PROGRAM FermentationProcess
VAR
	
(************** NAPĘDY **************************************************)
	fbDrv_MX01 		 : FB_Drive_1C();		//Napedy U11 mieszadła MX01	
	fbDrvContr_MX01  : FB_DriveControl(fbDrv_MX01);

	fbDrv_MX02 		 : FB_Drive_1C(); 		//Napedy U11 mieszadła MX01	
	fbDrvContr_MX02  : FB_DriveControl(fbDrv_MX02);

(************** Temp Sensor **************************************************)
	fbTempSens_T01	 : FB_Scaling; //Czujnik temperatury w reaktorze R01
	
(************** Ph Sensor **************************************************)
	fbPhSens_Ph01	 : FB_Scaling; //Czujnik ph w reaktorze R01

(************** Pressure Sensor **************************************************)
	fbPressureSens_P01	 : FB_Scaling; //Czujnik ciśnienia w reaktorze R01

(************** Hydrostatic pressure Sensor ************************************)
	fbHydrosPressureSens_HP01	  : FB_Scaling;
	
(************** Level Sensor **************************************************)
	fbLevelSens_L01	 : FB_Scaling; //Czujnik poziomu cieczy w reaktorze R01

(************** Reactor Mixers ***********************************************)
	fbReactorMixers	 : FB_ReactorMixer;	
	

END_VAR
VAR // added by the converter: edge detectors and wires of the graphical bodies
    _w1 : TIME;
    _w2 : ANY;
END_VAR

//Action
ACT_PhSens();       //skalowanie ph
ACT_PressureSens(); //skalowanie ciśnienie
ACT_TempSens();     //skalowanie temperatura
ACT_LevelSens();    //skalowanie poziom
ACT_Motor();    	//nastawy z SCADA
ACT_ReactorMixers();//Mieszanie w R01



//MX01
fbDrvContr_MX01();
GVL_Fermentation.stDriveStatus_MX01 := fbDrvContr_MX01.StatusStruct(); //zwróc strukturę

//MX02
fbDrvContr_MX02();
GVL_Fermentation.stDriveStatus_MX02 := fbDrvContr_MX02.StatusStruct(); //zwróc strukturę

ACTION ACT_LevelSens:
//Wyznacz poziom płynu w komorze fermentora zgodnie z wzorem (mH2O-P[kPa]*0.1)+poziom na ktorym wisi sonda hydrostatyczna
//przyjeto Ro =1kg/m3 g=9.81m2/s
GVL_Fermentation.LevelSens_R01.rValue := GVL_Fermentation.HydroPressSens_R01.rValue - GVL_Fermentation.PressureSens_R01.rValue * 0.1 + 0.12;
END_ACTION

ACTION ACT_Motor:
//Naped ustawienia MX01 i MX02
//nastawy z SCADA MX01
fbDrvContr_MX01.SetForward:=GVL_Fermentation.stDriveStatus_MX01.bForward;
//nastawy z SCADA MX02
fbDrvContr_MX02.SetForward:=GVL_Fermentation.stDriveStatus_MX02.bForward;
END_ACTION

ACTION ACT_PhSens:
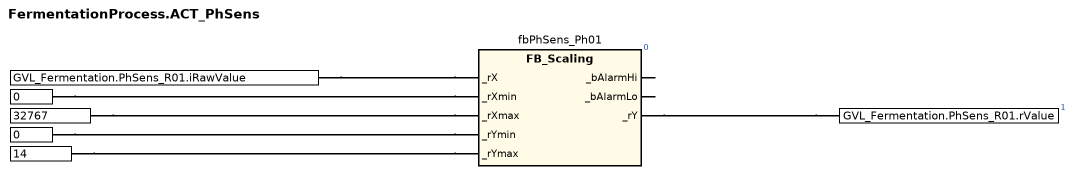
fbPhSens_Ph01(
    _rX := GVL_Fermentation.PhSens_R01.iRawValue,
    _rXmin := 0,
    _rXmax := 32767,
    _rYmin := 0,
    _rYmax := 14); // FB_Scaling
GVL_Fermentation.PhSens_R01.rValue := fbPhSens_Ph01._rY;
END_ACTION

ACTION ACT_PressureSens:
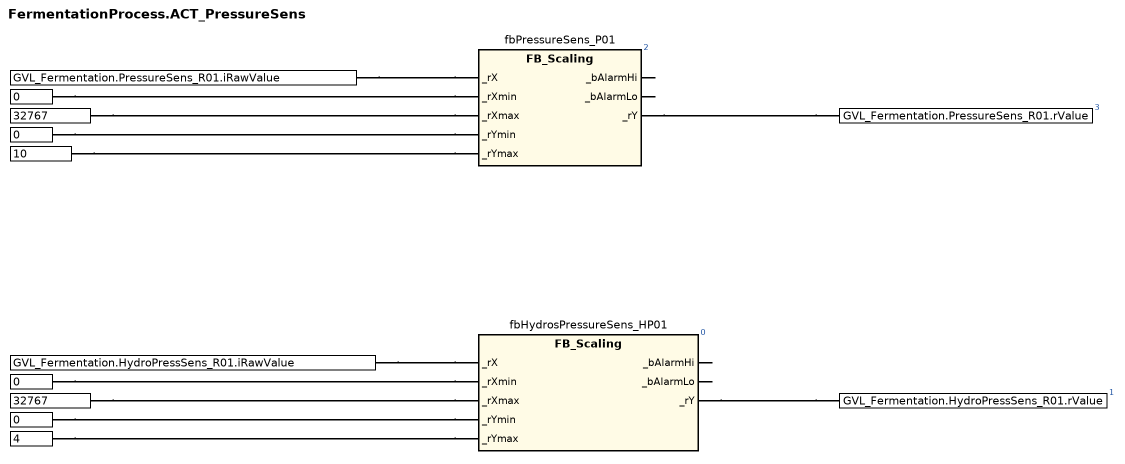
fbHydrosPressureSens_HP01(
    _rX := GVL_Fermentation.HydroPressSens_R01.iRawValue,
    _rXmin := 0,
    _rXmax := 32767,
    _rYmin := 0,
    _rYmax := 4); // FB_Scaling
GVL_Fermentation.HydroPressSens_R01.rValue := fbHydrosPressureSens_HP01._rY;
fbPressureSens_P01(
    _rX := GVL_Fermentation.PressureSens_R01.iRawValue,
    _rXmin := 0,
    _rXmax := 32767,
    _rYmin := 0,
    _rYmax := 10); // FB_Scaling
GVL_Fermentation.PressureSens_R01.rValue := fbPressureSens_P01._rY;
END_ACTION

ACTION ACT_ReactorMixers:
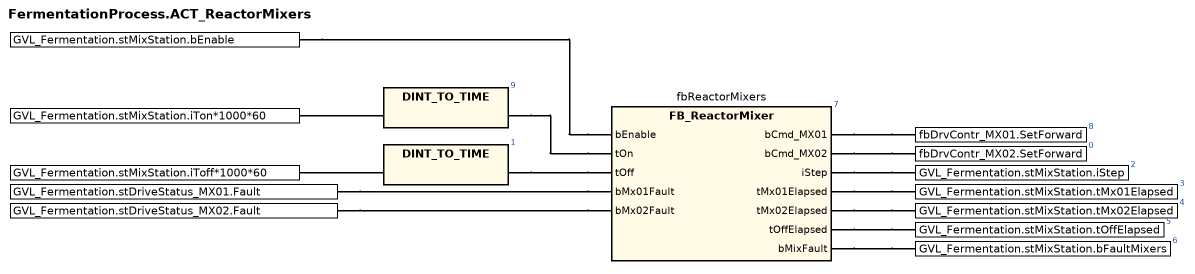
fbDrvContr_MX02.SetForward := fbReactorMixers.bCmd_MX02;
_w1 := DINT_TO_TIME(GVL_Fermentation.stMixStation.iToff*1000*60);
GVL_Fermentation.stMixStation.iStep := fbReactorMixers.iStep;
GVL_Fermentation.stMixStation.tMx01Elapsed := fbReactorMixers.tMx01Elapsed;
GVL_Fermentation.stMixStation.tMx02Elapsed := fbReactorMixers.tMx02Elapsed;
GVL_Fermentation.stMixStation.tOffElapsed := fbReactorMixers.tOffElapsed;
GVL_Fermentation.stMixStation.bFaultMixers := fbReactorMixers.bMixFault;
fbReactorMixers(
    bEnable := GVL_Fermentation.stMixStation.bEnable,
    tOn := _w2,
    tOff := _w1,
    bMx01Fault := GVL_Fermentation.stDriveStatus_MX01.Fault,
    bMx02Fault := GVL_Fermentation.stDriveStatus_MX02.Fault); // FB_ReactorMixer
fbDrvContr_MX01.SetForward := fbReactorMixers.bCmd_MX01;
_w2 := DINT_TO_TIME(GVL_Fermentation.stMixStation.iTon*1000*60);
END_ACTION

ACTION ACT_TempSens:
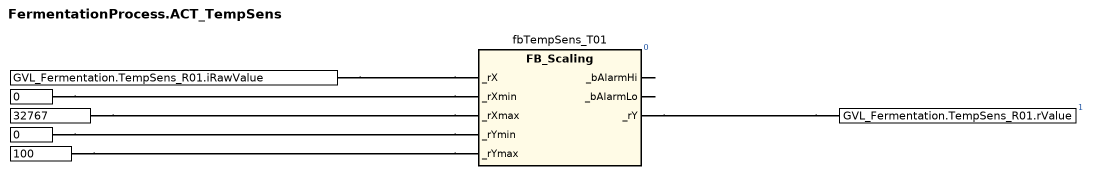
fbTempSens_T01(
    _rX := GVL_Fermentation.TempSens_R01.iRawValue,
    _rXmin := 0,
    _rXmax := 32767,
    _rYmin := 0,
    _rYmax := 100); // FB_Scaling
GVL_Fermentation.TempSens_R01.rValue := fbTempSens_T01._rY;
END_ACTION

END_PROGRAM

(* stored: Version 1.1.0.1, ProductVersion 3.1.4024.15
   POU FermentationProcess: Id {553c9373-2315-45e5-ad38-9104f2f846ac}, SpecialFunc None
   Action ACT_LevelSens: Id {5aba7613-72d4-4290-9316-0bee355161b2}
   Action ACT_Motor: Id {8b1ba2b0-5de3-4317-90d1-d6c08d7f8f90}
   Action ACT_PhSens: Id {8fd24e1d-da86-485b-b785-e45b2c1503a8}
   Action ACT_PressureSens: Id {cd1bc4d7-f2d8-49ae-a6ca-74cbcfd4394e}
   Action ACT_ReactorMixers: Id {a96e26f3-ffe2-4661-bf65-d9b1e8c251ad}
   Action ACT_TempSens: Id {9fdbb046-bcd0-4d84-b12c-c0b4c25c6026} *)
